(* Schneider Machine Expert - Basic project tank_level_v8_TM221CE24T, file version 3.0.0.0 *)
(* ProjectInformations: Name=New project *)

HARDWARE
  Cpu 0: TM221CE24T
  ModuleExtensionObject 0: TM3AI4/G
  EthernetConfiguration: NetworkName=M221, IpAllocationMode=FixedAddress, IpAddress=0.0.0.0, SubnetMask=0.0.0.0
  SerialLineConfiguration: Baud=Baud19200, Parity=ParityEven, DataBits=DataBits8, StopBits=StopBits1, PhysicalMedium=PhysicalMediumRs485, TransmissionMode=TransmissionModeModbusRtu, SlaveId=1, Addressing=SlaveAddressing
  MastTask: UsePeriodScanMode=false, PeriodScan=100
  FastTask: Period=255
  CpuBehavior: StartingMode=StartAsPreviousState, AutoSaveRamOnEeprom=true, WatchdogPeriod=250

SYMBOLS  (address, symbol, comment, settings)
  %S12      SB_RUNMODE  "The controller is running"
  %IW1.0    TANK_LEVEL  [Type=Type_4_20mA, Scope=Scope_Customized, Minimum=300, Maximum=3000]

POU Tank_Level_Control
  (* SectionNumber=0 *)

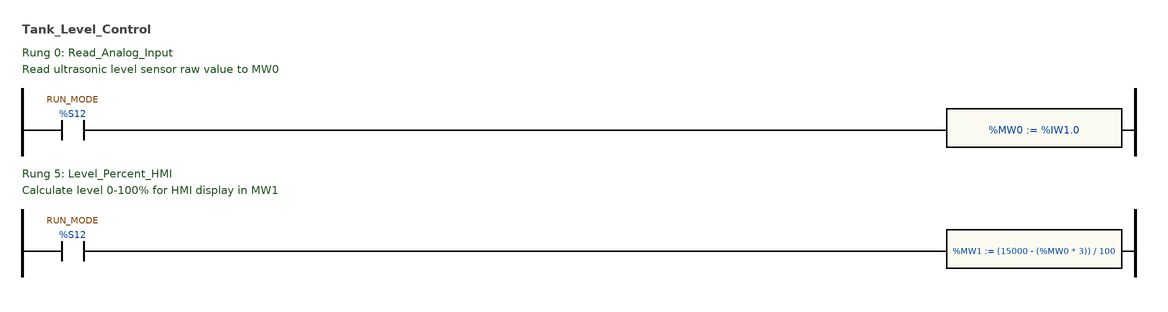

// Rung 0: Read_Analog_Input
// Read ultrasonic level sensor raw value to MW0
  LD %S12                 (* SB_RUNMODE *)
  [ %MW0 := %IW1.0 ]      (* TANK_LEVEL *)
  // as ST:
  //   IF SB_RUNMODE THEN %MW0 := TANK_LEVEL; END_IF;

// Rung 1: Tank_Full_Detection
// Tank FULL when raw less than 1800 (distance 540mm)
  LD [%MW0<1800]
  ST %M1
  // as ST:
  //   %M1 := %MW0<1800;
  (* the ladder stored for this rung does not match its IL; not drawn *)

// Rung 2: Tank_Empty_Detection
// Tank EMPTY when raw greater than 4800 (distance 1440mm)
  LD [%MW0>4800]
  ST %M2
  // as ST:
  //   %M2 := %MW0>4800;
  (* the ladder stored for this rung does not match its IL; not drawn *)

// Rung 3: Inlet_Valve_Control
// Hysteresis: Fill when empty, stop when full
  LD %M2
  OR %Q0.0
  ANDN %M1
  ST %Q0.0
  // as ST:
  //   %Q0.0 := (%M2 OR %Q0.0) AND NOT %M1;
  (* the ladder stored for this rung does not match its IL; not drawn *)

// Rung 4: Outlet_Valve_Control
// Hysteresis: Drain when full, stop when empty
  LD %M1
  OR %Q0.1
  ANDN %M2
  ST %Q0.1
  // as ST:
  //   %Q0.1 := (%M1 OR %Q0.1) AND NOT %M2;
  (* the ladder stored for this rung does not match its IL; not drawn *)

// Rung 5: Level_Percent_HMI
// Calculate level 0-100% for HMI display in MW1
  LD %S12                 (* SB_RUNMODE *)
  [ %MW1 := (15000 - (%MW0 * 3)) / 100 ]
  // as ST:
  //   IF SB_RUNMODE THEN %MW1 := (15000 - (%MW0 * 3)) / 100; END_IF;
